# EPICS autosave request: iocBoot/ioc13bmd_linux/auto_positions.req
file "Galil_positions.req", P=$(P)
